PROGRAM MAIN
VAR

END_VAR

drives();
P_TextModeWrite();

END_PROGRAM

(* stored: Version 1.1.0.1, ProductVersion 3.1.4024.12
   POU MAIN: Id {8c1c8652-12a0-4c66-a80d-55b797948f91}, SpecialFunc None *)
